{attribute 'GeneratedUsingTerminal: EL2262-0000-0001'}
{attribute addProperty BoxType "EL2262-0000-0001"}
{attribute addProperty Id "Cycle_CounterAT %Q*UINT2"}
{attribute addProperty CRC "740505604"}
{attribute addProperty Size "2"}
TYPE CycCount1_2C233804 EXTENDS OutputBase_10CEE7DE :
STRUCT
	{attribute addProperty Name "Cycle_Counter"}
	Cycle_Counter AT %Q* : UINT;
END_STRUCT
END_TYPE

(* stored: Version 1.2.0.0, ProductVersion 3.1.4024.9
   DUT CycCount1_2C233804: Id {d6499046-62db-409b-b9d2-cc7742aa7534} *)
